// TwinCAT 3 PLC project MONETRoof
// Title: MONET Roof
// Company: Georg-August-Universitaet Goettingen
// ProjectVersion: 1.1.5
// ProgramVersion: 3.1.4026.11
// libraries:
//   Tc2_Standard, * (Beckhoff Automation GmbH)
//   Tc2_System, * (Beckhoff Automation GmbH)
//   Tc3_Module, * (Beckhoff Automation GmbH)
//   BROTLib,newest,BROT
//   VisuSymbols,3.5.10.0,System
// project tree:
//   / GlobalTextList.TcGTLO, VisualizationManager.TcVMO (not stored)
//   POUs/ FB_Roof.TcPOU, FB_RoofControl.TcPOU, FB_RoofMotor.TcPOU, FB_Ramp.TcPOU
//   VISUs/ Roof.TcVIS
//   GVLs/ Global_Version.TcGVL

// ---- GVLs/Global_Version.TcGVL
{attribute 'qualified_only'}
VAR_GLOBAL CONSTANT
	// Mirrors Beckhoff's own Global_Version.stLibVersion_* pattern (see ST_LibVersion),
	// which only covers Tc2_*/Tc3_* library references, not custom ones -- until now: this
	// GVL uses Beckhoff's own naming exactly, so it merges into a consumer's Global_Version.
	// Kept in sync with <ProjectVersion> in MonetRoof.plcproj at release time.
	stLibVersion_MONETRoof : ST_LibVersion := (
		iMajor := 1,
		iMinor := 1,
		iBuild := 5,
		iRevision := 0,
		nFlags := 1,
		sVersion := '1.1.5'
	);
END_VAR

// ---- POUs/FB_Roof.TcPOU
FUNCTION_BLOCK FB_Roof
VAR_INPUT
	roof_number				: UINT;		// number of roof
	min_speed				: UINT;		// minimum speed to drive
	max_speed				: UINT;		// maximum speed to drive
	acceleration			: UINT;		// acceleration [speed/call]: the ramp time depends on the task cycle time (10 ms in all projects)
	min_position			: INT;		// minimum position of roof
	max_position			: INT;		// maximum position of roof
	max_position_diff		: INT;		// position difference between the two drives of the roof at which sync_error / limit_error trigger (smaller is tolerated)
	overtravel_margin		: INT := 10;	// stop if a drive counts more than this beyond min/max_position, e.g. with failed limit switches
	stall_timeout			: TIME := T#10S;	// stop if a drive is driven this long without a counter edge (see FB_RoofMotor)
	limit_slowdown			: REAL := 5;	// linear slowdown when moving towards limits starting at <x% and >(100-x)%
	comm					: I_Comm;
	reset_roof				: BOOL;

	slow_open				: BOOL := FALSE;	// open at min_speed, ignoring all errors and other commands
	slow_close				: BOOL := FALSE;	// close at min_speed, ignoring all errors and other commands
	
	zero_counter			: BOOL := FALSE;	// reset position counter of both motors to zero
END_VAR
VAR_OUTPUT
	sync_error				: BOOL;
	limit_error				: BOOL;
	overtravel_error		: BOOL;
	stall_error				: BOOL;
	drive_error				: BOOL;
	config_error			: BOOL;		// invalid parameters (speed / position range, max_position_diff, acceleration): the roof is held at 0
	state					: E_RoofState := E_RoofState.unknown;
	percent_open			: REAL;
	is_open					: BOOL;		// fully open (both open limit switches)
	is_closed				: BOOL;		// fully closed (both closed limit switches)
END_VAR
VAR_OUTPUT PERSISTENT
	position_valid			: BOOL;		// position counters are trustworthy: set by a limit snap, cleared by zero_counter and whenever the counters are lost
END_VAR
VAR
	// commands for roofs
	open_roof		AT%I*	: BOOL;
	close_roof		AT%I*	: BOOL;

	motors			: ARRAY[1..2] OF FB_RoofMotor;
	i				: UINT;
	
	roof_limit_open			: BOOL;		// whether any open limit switch for this roof is triggered
	roof_limit_closed		: BOOL;		// whether any close limit switch for this roof is triggered
	
	opened_event			: FB_EventLog;	// event for opened roof half
	closed_event			: FB_EventLog;	// event for closed roof half
	sync_error_event		: FB_EventLog;	// event for sync error
	limit_error_event		: FB_EventLog;	// event for limit error
	overtravel_error_event	: FB_EventLog;	// event for over-travel error
	stall_error_event		: FB_EventLog;	// event for stall error
	config_error_event		: FB_EventLog;	// event for configuration error
	
	// speed
	vel_ramp				: FB_Ramp;
	target_speed			: INT;	
	limit_speed				: REAL;
	speed					: INT;		// move speed
	
	// opening or closing?
	is_opening				: BOOL;		// move direction
	is_closing				: BOOL;	
	
	// boot-time snap guard
	bRoofInitialized		: BOOL;
END_VAR

// parameters that would make the speed wrap in TO_INT / UINT arithmetic, divide by zero in percent_open,
// or leave the roof with a permanent sync error or without any ramp
config_error := max_speed > 32767 OR min_speed > max_speed OR max_position <= min_position OR
				max_position_diff <= 0 OR acceleration = 0;

// limit switches for this roof?
roof_limit_open   := motors[1].opened AND motors[2].opened;
roof_limit_closed := motors[1].closed AND motors[2].closed;

// ramp for roof velocity (percent_open below is still the value from the end of the previous cycle)
IF slow_open THEN
	speed := TO_INT(min_speed); 
ELSIF slow_close THEN
	speed := -TO_INT(min_speed);
ELSE
	vel_ramp(
		start		:= speed,
		target		:= target_speed,
		accel		:= acceleration,
		value		=> speed);
END_IF

// get direction
is_opening := speed > 0;
is_closing := speed < 0;

// slowdown near limits
IF is_closing AND percent_open < limit_slowdown THEN
	// closing near limit
	IF percent_open <= 0 THEN
		limit_speed := -TO_INT(min_speed);
	ELSE
		limit_speed := -((percent_open / limit_slowdown) * (max_speed - min_speed) + min_speed);
	END_IF
	IF limit_speed > speed THEN
		speed :=  REAL_TO_INT(MAX(limit_speed, -TO_INT(max_speed)));
	END_IF	
END_IF
IF is_opening AND 100.0 - percent_open < limit_slowdown THEN
	// opening near limit
	IF percent_open >= 100 THEN
		limit_speed := min_speed;
	ELSE
		limit_speed := ((100.0 - percent_open) / limit_slowdown) * (max_speed - min_speed) + min_speed;
	END_IF
	IF limit_speed < speed THEN
		speed := REAL_TO_INT(MIN(limit_speed, max_speed));
	END_IF	
END_IF

// stop on limit switches
IF (is_closing AND roof_limit_closed) OR (is_opening AND roof_limit_open) THEN
	Stop();
END_IF

// boot-time position snap: warm restart with the roof parked at a limit.
// One-shot on the first cycle, both sensors together (symmetric — no |diff|).
// Uses FB_Roof's own min_position/max_position, not motors[i].min_position/max_position: the
// latter are FB_RoofMotor's VAR_INPUTs, only assigned by the motor call further below, so on the
// very first cycle ever (before that call has run once) they are still 0.
IF NOT bRoofInitialized THEN
	bRoofInitialized := TRUE;
	// position_valid is PERSISTENT and may be stale: TwinCAT does not flush persistent data every
	// cycle, so an uncontrolled power loss mid-move can restore a value from before the roof's last
	// recorded position, with position_valid still TRUE from that earlier, once-valid state. Distrust
	// it unconditionally on every restart (clean or not, there is no way to tell them apart here) and
	// require it to be reconfirmed below, exactly like a lost/zeroed counter.
	position_valid := FALSE;
	IF roof_limit_closed THEN
		motors[1].SetPosition(min_position);
		motors[2].SetPosition(min_position);
		position_valid := TRUE;
	ELSIF roof_limit_open THEN
		motors[1].SetPosition(max_position);
		motors[2].SetPosition(max_position);
		position_valid := TRUE;
	END_IF
END_IF

// limit re-sync: snap both drives to the physical end position (both sensors
// engaged). Direction-gated: must NOT fire at the START of a move while the
// opposite limit switch is still engaged (the first counter edge can arrive
// ~0.5 s before the closed switch releases) — an ungated snap would erase
// those legitimate counts and leave the move one count short. While stalled
// against a limit the snap holds the position, so stall-jitter counts cannot
// drive it past the end position.
IF is_closing AND roof_limit_closed THEN
	motors[1].SetPosition(min_position);
	motors[2].SetPosition(min_position);
	position_valid := TRUE;
END_IF
IF is_opening AND roof_limit_open THEN
	motors[1].SetPosition(max_position);
	motors[2].SetPosition(max_position);
	position_valid := TRUE;
END_IF

// zeroing the counters says nothing about where the roof is
IF zero_counter THEN
	position_valid := FALSE;
END_IF

// latched error: hold the drive at 0 from the start of the cycle. Without this a level command
// (button held, open_roofs set) re-arms the ramp every cycle and the drive gets one ramp step
// (real_speed = acceleration) before the error stop below zeroes it again.
// Slow mode ignores errors on purpose, so it is exempted here explicitly: it must not depend
// on the motors being called before the error stop.
// A configuration error is not exempted: with invalid parameters the speed can wrap to the
// opposite direction, slow mode included.
IF config_error OR (state = E_RoofState.error AND NOT slow_open AND NOT slow_close) THEN
	Stop();
END_IF

// call motors
drive_error := FALSE;
FOR i := 1 TO 2 DO
	// call individual motors
	motors[i](
		roof_number 		:= roof_number,
		drive_number 		:= i,
		min_position 		:= min_position, 
		max_position 		:= max_position,
		real_speed			:= speed,
		zero_counter		:= zero_counter,
		stall_timeout		:= stall_timeout,
		comm 				:= comm);
		
	// check errors
	IF motors[i].error THEN
		drive_error := TRUE;
	END_IF
END_FOR
percent_open := (motors[1].percent_open + motors[2].percent_open) / 2.0;

// fully open/closed
is_open := roof_limit_open;
is_closed := roof_limit_closed;

// consistency check: no direction_error any more (removed) — the two motors of a roof half are
// always called with the same speed and are mechanically coupled by a shaft, so they can never
// disagree on direction; a mismatch between them can only ever show up as sync_error.
sync_error := ABS(motors[1].position - motors[2].position) >= max_position_diff;
limit_error := (is_opening AND motors[1].MovedSinceOpen >= max_position_diff) OR 
			   (is_closing AND motors[1].MovedSinceClosed >= max_position_diff) OR
			   (is_opening AND motors[2].MovedSinceOpen >= max_position_diff) OR 
			   (is_closing AND motors[2].MovedSinceClosed >= max_position_diff);

// no software end stop otherwise: with failed limit switches nothing bounds the travel.
// Only while the position is known: after lost/zeroed counters (e.g. a reset with the roof
// halfway open) it would block moving towards the end the counters wrongly claim to be at.
overtravel_error := position_valid AND
					((is_opening AND (motors[1].position > max_position + overtravel_margin OR 
									  motors[2].position > max_position + overtravel_margin)) OR
					 (is_closing AND (motors[1].position < min_position - overtravel_margin OR 
									  motors[2].position < min_position - overtravel_margin)));

// a drive that is driven but does not count (jam, ice, dead sensor)
stall_error := motors[1].stall_error OR motors[2].stall_error;

// stop on error
IF sync_error OR drive_error OR limit_error OR overtravel_error OR stall_error OR config_error OR state = E_RoofState.error THEN
	Stop();
END_IF

// set state
IF sync_error OR drive_error OR limit_error OR overtravel_error OR stall_error OR config_error THEN
	state := E_RoofState.error;
ELSE
	// no current error, but if we're still in error state, only proceed, if reset_roof is set
	IF state <> E_RoofState.error OR reset_roof THEN
		reset_roof := FALSE; 	

		// check other states
		// both motors get the same speed, so a moving roof has exactly one direction
		IF motors[1].moving OR motors[2].moving THEN
			IF motors[1].direction_open OR motors[2].direction_open THEN
				state := E_RoofState.opening;
			ELSE
				state := E_RoofState.closing;
			END_IF
		ELSIF roof_limit_open THEN
			// fully open needs both switches, like is_open; one switch alone is only 'stopped'
			state := E_RoofState.opened;
		ELSIF roof_limit_closed THEN
			state := E_RoofState.closed;
		ELSE
			state := E_RoofState.stopped;
		END_IF
	END_IF
END_IF

// events
opened_event(
	Trigger := is_open, 
	Level := ADSLOG_MSGTYPE_HINT, 
	FormatString := 'Roof #%s is fully open.', 
	OnMessage := UINT_TO_STRING(roof_number),
	Comm := comm);
closed_event(
	Trigger := is_closed, 
	Level := ADSLOG_MSGTYPE_HINT, 
	FormatString := 'Roof #%s is fully closed.', 
	OnMessage := UINT_TO_STRING(roof_number),
	Comm := comm); 

// errors
sync_error_event(
	Trigger := sync_error, 
	Level := ADSLOG_MSGTYPE_ERROR, 
	FormatString := 'Drives for roof #%s out of sync.', 
	OnMessage := UINT_TO_STRING(roof_number),
	Comm := comm); 
limit_error_event(
	Trigger := limit_error, 
	Level := ADSLOG_MSGTYPE_ERROR, 
	FormatString := 'Could not find 2nd limit switch for roof #%s.', 
	OnMessage := UINT_TO_STRING(roof_number),
	Comm := comm); 
overtravel_error_event(
	Trigger := overtravel_error, 
	Level := ADSLOG_MSGTYPE_ERROR, 
	FormatString := 'Roof #%s moved beyond its end position.', 
	OnMessage := UINT_TO_STRING(roof_number),
	Comm := comm); 
stall_error_event(
	Trigger := stall_error, 
	Level := ADSLOG_MSGTYPE_ERROR, 
	FormatString := 'Drive of roof #%s does not move (no counts).',
	OnMessage := UINT_TO_STRING(roof_number),
	Comm := comm);
config_error_event(
	Trigger := config_error,
	Level := ADSLOG_MSGTYPE_ERROR,
	FormatString := 'Roof #%s has invalid parameters.',
	OnMessage := UINT_TO_STRING(roof_number),
	Comm := comm);

METHOD Automatic : BOOL
VAR_INPUT
	open_roof	: BOOL;
	close_roof	: BOOL;
	stop_roof	: BOOL;
END_VAR
// automatic commands 
IF open_roof THEN
	Open();
ELSIF close_roof THEN
	Close();
ELSIF stop_roof THEN
	SoftStop();
END_IF
END_METHOD

METHOD Close : BOOL
VAR_INPUT
END_VAR
IF NOT slow_open AND NOT slow_close THEN
	IF NOT is_closed THEN
		target_speed := -TO_INT(max_speed);
	END_IF
END_IF
END_METHOD

PROPERTY Error : STRING
GET
// invalid parameters come first, the other checks are meaningless with them;
// then a drive fault: it is usually the root cause of the stall or sync error that follows
IF config_error THEN
	Error := 'Configuration error';
ELSIF drive_error THEN
	Error := 'Drive error';
ELSIF sync_error THEN
	Error := 'Sync error';
ELSIF limit_error THEN
	Error := 'Limit error';
ELSIF overtravel_error THEN
	Error := 'Over-travel error';
ELSIF stall_error THEN
	Error := 'Stall error';
ELSE
	Error := '';
END_IF
END_GET
END_PROPERTY

METHOD Manual : BOOL
VAR_INPUT
END_VAR
// manual commands commands
IF open_roof THEN
	Open();
ELSIF close_roof THEN
	Close();
ELSE
	SoftStop();
END_IF
END_METHOD

METHOD Open : BOOL
VAR_INPUT
END_VAR
VAR
END_VAR
IF NOT slow_open AND NOT slow_close THEN
	IF NOT is_open THEN
		target_speed := TO_INT(max_speed);
	END_IF
END_IF
END_METHOD

METHOD Reset : BOOL
VAR_INPUT
END_VAR
reset_roof := TRUE;
FOR i := 1 TO 2 DO
	motors[i].Reset();
END_FOR;
END_METHOD

METHOD SoftStop : BOOL
VAR_INPUT
END_VAR
target_speed := 0;
END_METHOD

PROPERTY Status : STRING
GET
IF state = E_RoofState.closed THEN
	Status := 'CLOSED';
ELSIF state = E_RoofState.opened THEN
	Status := 'OPENED';
ELSIF state = E_RoofState.opening THEN
	Status := 'OPENING';
ELSIF state = E_RoofState.closing THEN
	Status := 'CLOSING';
ELSIF state = E_RoofState.stopped THEN
	Status := 'STOPPED';
ELSIF state = E_RoofState.error THEN
	Status := 'ERROR';
ELSIF state = E_RoofState.unknown THEN
	Status := 'UNKNOWN';	
END_IF
END_GET
END_PROPERTY

METHOD Stop : BOOL
VAR_INPUT
END_VAR
speed := 0;
target_speed := 0;
END_METHOD

END_FUNCTION_BLOCK

// ---- POUs/FB_RoofMotor.TcPOU
FUNCTION_BLOCK FB_RoofMotor
VAR_INPUT
	roof_number				: UINT;		// number of roof
	drive_number			: UINT;		// number of drive
	min_position			: INT;		// minimum position of roof
	max_position			: INT;		// maximum position of roof
	real_speed				: INT;		// signed speed
	zero_counter			: BOOL := FALSE;	// reset position counter to zero
	comm					: I_Comm;
	
	// counting filters (insurance; defaults sized from the recordings — plan 2026-08-20)
	counter_debounce		: TIME := T#5MS;	// min. on-time of a sensor pulse. Keep clear of the 10 ms task cycle: at
										// PT = cycle time, ordinary cycle jitter can push the elapsed time on the
										// deciding scan just under PT and drop an otherwise-valid pulse entirely
										// (modelled in testing/check_debounce_aliasing.py). 5 ms sits above the
										// EL1008's ~3 ms input filter and comfortably below one cycle.
	counter_min_spacing		: TIME := T#50MS;	// min. time between accepted counts — keep < rotation period (600 ms)
	
	// stall watchdog
	stall_timeout			: TIME := T#10S;	// max. time moving without an accepted count — keep well above the rotation period (0.6 s at max_speed, slower at min_speed) and the ~3 s until the first count after a start
END_VAR
VAR_OUTPUT PERSISTENT
	position				: INT;	// position
END_VAR
VAR_OUTPUT
	percent_open			: REAL;	// percentage open
	
	// moving
	moving					: BOOL;
	
	// debug: raw (unfiltered, ungated) edge count for validation
	raw_counts				: DINT;
	
	// error 
	motor_error		AT%I*	: BOOL;
	error					: BOOL;
	stall_error				: BOOL;	// moving, but no counter edge for stall_timeout (jammed drive, dead sensor)
	
	// signals from limit switches
	opened			AT%I*	: BOOL;
	closed			AT%I*	: BOOL;
	
	// position on limit switch
	position_open			: INT := -1000;
	position_close			: INT := -1000;
END_VAR
VAR
	// error
	drive_error_event		: FB_EventLog;

	// inductive sensor for counting rotation
	counter			AT%I*	: BOOL;
	counter_trig			: R_TRIG;
	counter_raw_trig		: R_TRIG;	// raw (unfiltered) edge trigger — for validation only
	tonDebounce				: TON;		// level debounce for the sensor pulse
	tonSpacing				: TON;		// rate limit: min. spacing between accepted counts
	tonStall				: TON;		// time since the last accepted count while moving
	bCountAccepted			: BOOL;		// a count was accepted in this cycle
	
	// reset command to drive
	reset_command			: BOOL;
	reset_timer				: TON;
	reset_drive		AT%Q*	: BOOL;
	
	// speed
	speed			AT%Q*	: INT;		// move speed
	direction_open	AT%Q*	: BOOL;		// move direction
	direction_close	AT%Q*	: BOOL;
	
	// position on limit switch
	position_open_on_trig	: R_TRIG;
	position_open_off_trig	: F_TRIG;
	position_close_on_trig	: R_TRIG;
	position_close_off_trig	: F_TRIG;
END_VAR

// signals
error := NOT motor_error;

// reset?
//reset_timer();
IF reset_command THEN
	// set signal and start timer
	reset_drive := TRUE;
	reset_timer(IN := TRUE, PT := T#200MS);
END_IF
IF reset_timer.Q THEN
	// reset everything
	reset_drive := FALSE;
	reset_command := FALSE;
	reset_timer(IN := FALSE);
END_IF

// relative position; FB_Roof still calls the motors with max_position <= min_position when config_error is set,
// and a division by zero stops the user-mode runtime (STATUS_FLOAT_DIVIDE_BY_ZERO)
IF max_position > min_position THEN
	percent_open := 1.0 * (position - min_position) / (max_position - min_position) * 100.0;
ELSE
	percent_open := 0.0;
END_IF

// get direction
direction_open := real_speed > 0;
direction_close := real_speed < 0;

// set moving before the counter gate (motion gate: no counting while idle)
moving := real_speed <> 0;

// counter for position — filtered and gated.
// The limit re-sync in FB_Roof is the primary protection; these layers are
// insurance only. Deliberately NOT gated on the limit switches: that would
// blind the sync check to a broken connection or a stalled drive.
tonDebounce(IN := counter, PT := counter_debounce);	// stable-high filter (kills short glitches)
counter_trig(CLK := tonDebounce.Q);					// edge of the filtered signal

// raw edge count (unfiltered, ungated) — for validation/comparison
counter_raw_trig(CLK := counter);
IF counter_raw_trig.Q THEN
	raw_counts := raw_counts + 1;
END_IF

bCountAccepted := FALSE;
IF counter_trig.Q AND moving THEN					// motion gate
	IF tonSpacing.Q THEN							// spacing window since last accepted count elapsed -> accept
		tonSpacing(IN := FALSE);					// restart the spacing window
		bCountAccepted := TRUE;
		IF direction_open THEN
			position := position + 1;
		ELSIF direction_close THEN
			position := position - 1;
		END_IF
	END_IF
END_IF
tonSpacing(IN := TRUE, PT := counter_min_spacing);	// rate limit timer (runs continuously)

// stall watchdog: driven, but the position counter does not advance (both drives jammed
// gives no position difference, so sync_error cannot see it)
tonStall(IN := moving AND NOT bCountAccepted, PT := stall_timeout);
stall_error := tonStall.Q;

// zero?
IF zero_counter THEN
	position := 0;
	raw_counts := 0;
END_IF

// remember position when entering/leaving limit switches
position_open_on_trig(CLK := opened);
IF position_open_on_trig.Q THEN
	position_open := position;
END_IF
position_open_off_trig(CLK := opened);
IF position_open_off_trig.Q THEN
	position_open := -1000;
END_IF
position_close_on_trig(CLK := closed);
IF position_close_on_trig.Q THEN
	position_close := position;
END_IF
position_close_off_trig(CLK := closed);
IF position_close_off_trig.Q THEN
	position_close := -1000;
END_IF

// absolute speed
speed := ABS(real_speed);

// error
drive_error_event(	
	Trigger 		:= error, 
	Level 			:= ADSLOG_MSGTYPE_ERROR,
	FormatString 	:= 'Drive %s in error state.', 
	OnMessage 		:= CONCAT(CONCAT(CONCAT('#', UINT_TO_STRING(drive_number)), ' of roof #'), UINT_TO_STRING(roof_number)),
	Comm			:= comm);

PROPERTY MovedSinceClosed : INT
GET
IF position_close = -1000 THEN
	MovedSinceClosed := 0;
ELSE
	MovedSinceClosed := ABS(position - position_close);
END_IF
END_GET
END_PROPERTY

PROPERTY MovedSinceOpen : INT
GET
IF position_open = -1000 THEN
	MovedSinceOpen := 0;
ELSE
	MovedSinceOpen := ABS(position - position_open);
END_IF
END_GET
END_PROPERTY

METHOD Reset : BOOL
VAR_INPUT
END_VAR
reset_command := TRUE;
END_METHOD

METHOD SetPosition : BOOL
VAR_INPUT
	position_value		: INT;		// new position value (e.g. min/max_position on limit re-sync)
END_VAR
// 'position' is a VAR_OUTPUT — read-only from outside the FB, so the
// FB_Roof-level limit re-sync sets it through this method.
position := position_value;

// Re-anchor the limit-switch records of a switch that is engaged right now. They hold the counter
// reading at engagement, which is meaningless after the snap (e.g. a restart with the roof half
// open: the switch engages at a wrong reading, the snap then corrects the counter). Left alone,
// MovedSince* would report the correction as travel and raise a false limit_error.
// A drive that really overruns its switch still trips limit_error: that check runs every cycle
// before a snap can happen, and a snap needs both switches engaged.
IF opened THEN
	position_open := position_value;
END_IF
IF closed THEN
	position_close := position_value;
END_IF
END_METHOD

END_FUNCTION_BLOCK

// ---- POUs/FB_Ramp.TcPOU
FUNCTION_BLOCK FB_Ramp
VAR_INPUT
	start	: INT;
	target	: INT;
	accel	: UINT;
END_VAR
VAR_OUTPUT
	value	: INT;
END_VAR
VAR
END_VAR

value := start;

// step
// compare in DINT: a reversal (e.g. -30000 -> +30000) does not fit in 16 bit
IF TO_DINT(target) - TO_DINT(value) > 0 THEN	
	value := value + TO_INT(accel);
	IF value >= target THEN
		value := target;
	END_IF
ELSE
	value := value - TO_INT(accel);
	IF value <= target THEN
		value := target;
	END_IF
END_IF

END_FUNCTION_BLOCK

// ---- POUs/FB_RoofControl.TcPOU
FUNCTION_BLOCK FB_RoofControl IMPLEMENTS I_Roof
VAR_INPUT
	min_speed				: UINT;			// minimum speed to drive
	max_speed				: UINT;			// maximum speed to drive
	acceleration			: UINT;			// acceleration [speed/call]
	max_position_diff		: INT;			// position difference between the two drives of a roof at which sync_error / limit_error trigger (smaller is tolerated)
	limit_slowdown			: REAL := 5;	// linear slowdown when moving towards limits starting at <x% and >(100-x)%
	min_position_1			: INT := 0;		// minimum position of roof
	max_position_1			: INT := 200;		// maximum position of roof
	min_position_2			: INT := 0;		// minimum position of roof
	max_position_2			: INT := 200;		// maximum position of roof

	// commands for automatic roof controls
	open_roofs				: BOOL;
	close_roofs				: BOOL;
	stop_roofs				: BOOL;
	reset_roofs				: BOOL;	
	open_roof				: ARRAY[1..2] OF BOOL;
	close_roof				: ARRAY[1..2] OF BOOL;
	stop_roof				: ARRAY[1..2] OF BOOL;
	reset_roof				: ARRAY[1..2] OF BOOL;
	
	// automatic mode
	automatic		AT%I*	: BOOL;
	
	// UPS failure: linked to the UPS input in the consumer projects (tsproj), not evaluated yet
	ups_fail		AT%I*	: BOOL;
	
	// telemetry interval
	fTelemetryInterval		: TIME := T#5S;
END_VAR
VAR_OUTPUT
	// state
	roof_state				: E_RoofState;
	percent_open			: REAL;	
END_VAR
VAR
	// roofs
	roofs					: ARRAY[1..2] OF FB_Roof;
	
	// loop variable	
	i						: UINT;
	
	// open and close delays
	tonOpen2Delay			: TON;
	tonClose1Delay			: TON;
	
	// Comm
	fbComm					: I_Comm;	
	tonComm 				: TON;
	
	min_positions			: ARRAY[1..2] OF INT;		// minimum position of roof
	max_positions			: ARRAY[1..2] OF INT;		// maximum position of roof
END_VAR

// min_max
min_positions[1] := min_position_1;
max_positions[1] := max_position_1;
min_positions[2] := min_position_2;
max_positions[2] := max_position_2;

// call roofs
FOR i := 1 TO 2 DO
	// reset
	IF reset_roofs OR reset_roof[i] THEN
		roofs[i].Reset();
	END_IF	

	// automatic or manual mode
	IF automatic THEN
		roofs[i].Automatic(open_roof := open_roofs OR open_roof[i], close_roof := close_roofs OR close_roof[i], stop_roof := stop_roofs OR stop_roof[i]);
	ELSE
		roofs[i].Manual();
	END_IF

	// run 
	roofs[i](		
		roof_number			:= i,
		min_speed			:= min_speed,
		max_speed 			:= max_speed, 
		acceleration 		:= acceleration, 
		min_position 		:= min_positions[i], 
		max_position 		:= max_positions[i],
		max_position_diff 	:= max_position_diff,
		limit_slowdown		:= limit_slowdown,
		comm 				:= fbComm
	);
END_FOR

// set state
IF roofs[1].state = E_RoofState.error OR roofs[2].state = E_RoofState.error THEN
	roof_state := E_RoofState.error;
ELSIF roofs[1].state = E_RoofState.opened AND roofs[2].state = E_RoofState.opened THEN
	roof_state := E_RoofState.opened;
ELSIF roofs[1].state = E_RoofState.closed AND roofs[2].state = E_RoofState.closed THEN
	roof_state := E_RoofState.closed;
ELSIF roofs[1].state = E_RoofState.opening OR roofs[2].state = E_RoofState.opening THEN
	roof_state := E_RoofState.opening;	
ELSIF roofs[1].state = E_RoofState.closing OR roofs[2].state = E_RoofState.closing THEN
	roof_state := E_RoofState.closing;
ELSIF (roofs[1].state = E_RoofState.stopped OR roofs[1].state = E_RoofState.opened OR roofs[1].state = E_RoofState.closed) AND 
      (roofs[2].state = E_RoofState.stopped OR roofs[2].state = E_RoofState.opened OR roofs[2].state = E_RoofState.closed) THEN
	roof_state := E_RoofState.stopped;
ELSE
	roof_state := E_RoofState.error;	
END_IF

// percent open, clamped to 0..100: the over-travel margin and unsynced counters (after a restart with
// the roof halfway open) let the raw value leave that range, and telemetry uses -1.0 as the error marker.
// The per-roof values stay raw as a diagnostic of the counters.
percent_open := MAX(0.0, MIN(100.0, (roofs[1].percent_open + roofs[2].percent_open) / 2.0));

// send telemetry
tonComm(IN:=TRUE, PT:=fTelemetryInterval);
IF tonComm.Q THEN // publish new payload every fTelemetryInterval (default 5 seconds)
	tonComm(IN:=FALSE);
	THIS^._SendTelemetry();	
END_IF

METHOD _SendTelemetry : BOOL
VAR_INPUT
END_VAR
IF roof_state = E_RoofState.opened THEN
	fbComm.Publish('telescope', 'dome', 'AUXILIARY.DOME.REALPOS', '1.0');
ELSIF roof_state = E_RoofState.closed THEN
	fbComm.Publish('telescope', 'dome', 'AUXILIARY.DOME.REALPOS', '0.0');
ELSIF roof_state = E_RoofState.error THEN
	fbComm.Publish('telescope', 'dome', 'AUXILIARY.DOME.REALPOS', '-1.0');
ELSE
	fbComm.Publish('telescope', 'dome', 'AUXILIARY.DOME.REALPOS', LREAL_TO_STRING(percent_open / 100.0));
END_IF

IF roof_state = E_RoofState.opened OR roof_state = E_RoofState.opening THEN
	fbComm.Publish('telescope', 'dome', 'AUXILIARY.DOME.TARGETPOS', '1.0');
ELSIF roof_state = E_RoofState.closed OR roof_state = E_RoofState.closing THEN
	fbComm.Publish('telescope', 'dome', 'AUXILIARY.DOME.TARGETPOS', '0.0');
ELSIF roof_state = E_RoofState.stopped THEN
	fbComm.Publish('telescope', 'dome', 'AUXILIARY.DOME.TARGETPOS', LREAL_TO_STRING(percent_open / 100.0));
ELSE
	fbComm.Publish('telescope', 'dome', 'AUXILIARY.DOME.TARGETPOS', '-1.0');
END_IF

IF roof_state = E_RoofState.error THEN
	fbComm.Publish('telescope', 'dome', 'AUXILIARY.DOME.ERROR_STATE', '1');
	fbComm.Publish('telescope', 'dome', 'AUXILIARY.DOME.READY_STATE', '-1.0');
ELSE
	fbComm.Publish('telescope', 'dome', 'AUXILIARY.DOME.ERROR_STATE', '0');
	IF roof_state = E_RoofState.closed THEN
		fbComm.Publish('telescope', 'dome', 'AUXILIARY.DOME.READY_STATE', '0.0');
	ELSE
		fbComm.Publish('telescope', 'dome', 'AUXILIARY.DOME.READY_STATE', '1.0');
	END_IF
END_IF

IF state = E_RoofState.opening OR state = E_RoofState.closing THEN
	fbComm.Publish('telescope', 'dome', 'AUXILIARY.DOME.MOTION_STATE', '1.0');
ELSE
	fbComm.Publish('telescope', 'dome', 'AUXILIARY.DOME.MOTION_STATE', '0.0');
END_IF

// MONET specific
fbComm.Publish('telescope', 'dome', 'MONET.ROOF.STATE', Status);
fbComm.Publish('telescope', 'dome', 'MONET.ROOF.POS1', LREAL_TO_STRING(roofs[1].percent_open));
fbComm.Publish('telescope', 'dome', 'MONET.ROOF.STATE1', roofs[1].Status);
fbComm.Publish('telescope', 'dome', 'MONET.ROOF.ERROR1', roofs[1].Error);
fbComm.Publish('telescope', 'dome', 'MONET.ROOF.POS2', LREAL_TO_STRING(roofs[2].percent_open));
fbComm.Publish('telescope', 'dome', 'MONET.ROOF.STATE2', roofs[2].Status);
fbComm.Publish('telescope', 'dome', 'MONET.ROOF.ERROR2', roofs[2].Error);
END_METHOD

METHOD Close : BOOL
VAR_INPUT
END_VAR
FOR i := 1 TO 2 DO
	roofs[i].Close();
END_FOR;
END_METHOD

//FB_Init is always available implicitly and it is used primarily for initialization.
//The return value is not evaluated. For a specific influence, you can also declare the
//methods explicitly and provide additional code there with the standard initialization
//code. You can evaluate the return value.
METHOD FB_Init: BOOL
VAR_INPUT
    bInitRetains	: BOOL; // TRUE: the retain variables are initialized (reset warm / reset cold)
    bInCopyCode		: BOOL;  // TRUE: the instance will be copied to the copy code afterward (online change)
	comm			: I_Comm;   
END_VAR
THIS^.fbComm := comm;
END_METHOD

METHOD Open : BOOL
VAR_INPUT
END_VAR
FOR i := 1 TO 2 DO
	roofs[i].Open();
END_FOR;
END_METHOD

METHOD Reset : BOOL
VAR_INPUT
END_VAR
FOR i := 1 TO 2 DO
	roofs[i].Reset();
END_FOR;
END_METHOD

PROPERTY State : E_RoofState
GET
State := roof_state;
END_GET
END_PROPERTY

PROPERTY Status : STRING
GET
IF state = E_RoofState.closed THEN
	Status := 'CLOSED';
ELSIF state = E_RoofState.opened THEN
	Status := 'OPENED';
ELSIF state = E_RoofState.opening THEN
	Status := 'OPENING';
ELSIF state = E_RoofState.closing THEN
	Status := 'CLOSING';
ELSIF state = E_RoofState.stopped THEN
	Status := 'STOPPED';
ELSIF state = E_RoofState.error THEN
	Status := 'ERROR';
ELSIF state = E_RoofState.unknown THEN
	Status := 'UNKNOWN';	
END_IF
END_GET
END_PROPERTY

METHOD Stop : BOOL
VAR_INPUT
END_VAR
FOR i := 1 TO 2 DO
	roofs[i].Stop();
END_FOR;
END_METHOD

END_FUNCTION_BLOCK

// ---- GlobalTextList.TcGTLO
TEXTLIST GlobalTextList
  265 = '%.0f %'
  194 = '%.2f'
  616 = '%d'
  606 = '%d %'
  759 = '%d %%'
  792 = '%s'
  148 = 'Automatic'
  337 = 'Close'
  507 = 'Closed'
  272 = 'Closing'
  937 = 'Dir Error'
  59 = 'Directio n Error'
  475 = 'Direction Error'
  957 = 'Direction error'
  511 = 'Drive   Error'
  264 = 'DriveError'
  298 = 'Error'
  389 = 'Motor #1'
  611 = 'Motor #2'
  765 = 'Moving'
  576 = 'None'
  366 = 'Open'
  186 = 'Opening'
  523 = 'Position'
  375 = 'Reset'
  798 = 'Roof'
  456 = 'Roof #1'
  944 = 'Roof #2'
  138 = 'Slow close'
  996 = 'Slow open'
  49 = 'Speed'
  520 = 'State'
  838 = 'Stop'
  790 = 'Stopped'
  619 = 'Sync Error'
  385 = 'Sync error'
  609 = 'Zero counter'
END_TEXTLIST

// ---- VISUs/Roof.TcVIS
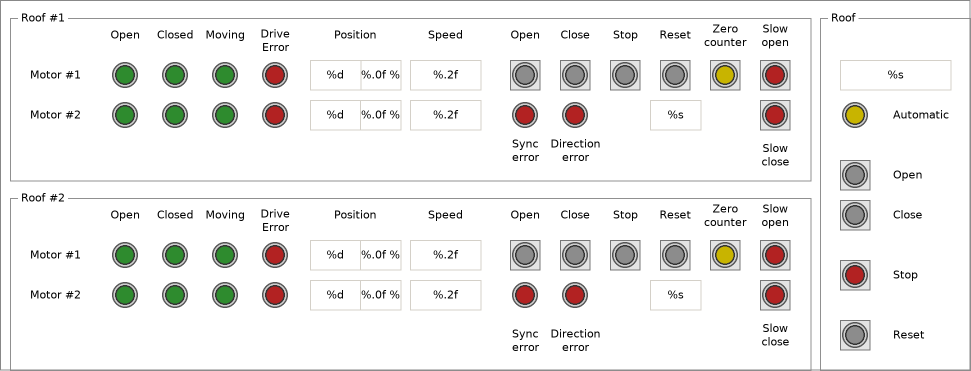
VISUALIZATION Roof  // 971x371
    GroupBox (10,10 801x171), "Roof #1"
        Label (10,50 71x30), "Motor #1"
        Label (10,90 71x30), "Motor #2"
        Label (80,10 71x30), "Open"
        Label (130,10 71x30), "Closed"
        Lamp1 (100,50 30x30), variable: MAIN.RoofControl.roofs[1].motors[1].opened, style: Lamp-Lamp1-Green
        Lamp1 (150,50 30x30), variable: MAIN.RoofControl.roofs[1].motors[1].closed, style: Lamp-Lamp1-Green
        Lamp1 (100,90 30x30), variable: MAIN.RoofControl.roofs[1].motors[2].opened, style: Lamp-Lamp1-Green
        Lamp1 (150,90 30x30), variable: MAIN.RoofControl.roofs[1].motors[2].closed, style: Lamp-Lamp1-Green
        Label (180,10 71x30), "Moving"
        Lamp1 (200,50 30x30), variable: MAIN.RoofControl.roofs[1].motors[1].moving, style: Lamp-Lamp1-Green
        Lamp1 (200,90 30x30), variable: MAIN.RoofControl.roofs[1].motors[2].moving, style: Lamp-Lamp1-Green
        Label (310,10 71x30), "Position"
        Textfield (350,50 41x30), "%.0f %", text variable: MAIN.RoofControl.roofs[1].motors[1].percent_open, input disabled if: TRUE
        Textfield (300,90 51x30), "%d", text variable: MAIN.RoofControl.roofs[1].motors[2].position, input disabled if: TRUE
        Label (400,10 71x30), "Speed"
        Textfield (400,50 71x30), "%.2f", text variable: MAIN.RoofControl.roofs[1].motors[1].speed, input disabled if: TRUE
        Textfield (400,90 71x30), "%.2f", text variable: MAIN.RoofControl.roofs[1].motors[2].speed, input disabled if: TRUE
        Label (480,10 71x30), "Open"
        PushSwitch (500,50 30x30), variable: MAIN.RoofControl.open_roof[1], behaviour: TAP, style: Switch-PushSwitch-Gray
        PushSwitch (550,50 30x30), variable: MAIN.RoofControl.close_roof[1], behaviour: TAP, style: Switch-PushSwitch-Gray
        Label (530,10 71x30), "Close"
        Label (590,10 51x30), "Stop"
        PushSwitch (600,50 30x30), variable: MAIN.RoofControl.stop_roof[1], behaviour: TAP, style: Switch-PushSwitch-Gray
        Lamp1 (500,90 30x30), variable: MAIN.RoofControl.roofs[1].sync_error, style: Lamp-Lamp1-Red
        Textfield (640,90 51x30), "%s", text variable: MAIN.RoofControl.roofs[1].state, input disabled if: TRUE
        Textfield (300,50 51x30), "%d", text variable: MAIN.RoofControl.roofs[1].motors[1].position, input disabled if: TRUE
        Textfield (350,90 41x30), "%.0f %", text variable: MAIN.RoofControl.roofs[1].motors[2].percent_open, input disabled if: TRUE
        Label (240,10 51x41), "Drive Error"
        Lamp1 (550,90 30x30), variable: MAIN.RoofControl.roofs[1].direction_error, style: Lamp-Lamp1-Red
        Label (490,120 51x41), "Sync error"
        Label (530,120 71x41), "Direction error"
        Label (640,10 51x30), "Reset"
        Lamp1 (250,50 30x30), variable: MAIN.RoofControl.roofs[1].motors[1].error, style: Lamp-Lamp1-Red
        Lamp1 (250,90 30x30), variable: MAIN.RoofControl.roofs[1].motors[2].error, style: Lamp-Lamp1-Red
        PushSwitch (750,50 30x30), variable: MAIN.RoofControl.roofs[1].slow_open, behaviour: TAP, style: Switch-PushSwitch-Red
        Label (740,10 51x31), "Slow open"
        Label (740,130 51x30), "Slow close"
        PushSwitch (750,230 30x30), variable: MAIN.RoofControl.stop_roof[1], behaviour: TAP, style: Switch-PushSwitch-Gray
        Label (690,10 51x31), "Zero counter"
    GroupBox (10,190 801x181), "Roof #2"
        Label (10,50 71x30), "Motor #1"
        Label (10,90 71x30), "Motor #2"
        Label (80,10 71x30), "Open"
        Label (130,10 71x30), "Closed"
        Lamp1 (100,50 30x30), variable: MAIN.RoofControl.roofs[2].motors[1].opened, style: Lamp-Lamp1-Green
        Lamp1 (150,50 30x30), variable: MAIN.RoofControl.roofs[2].motors[1].closed, style: Lamp-Lamp1-Green
        Lamp1 (100,90 30x30), variable: MAIN.RoofControl.roofs[2].motors[2].opened, style: Lamp-Lamp1-Green
        Lamp1 (150,90 30x30), variable: MAIN.RoofControl.roofs[2].motors[2].closed, style: Lamp-Lamp1-Green
        Label (180,10 71x30), "Moving"
        Lamp1 (200,50 30x30), variable: MAIN.RoofControl.roofs[2].motors[1].moving, style: Lamp-Lamp1-Green
        Lamp1 (200,90 30x30), variable: MAIN.RoofControl.roofs[2].motors[2].moving, style: Lamp-Lamp1-Green
        Label (310,10 71x30), "Position"
        Textfield (300,50 51x30), "%d", text variable: MAIN.RoofControl.roofs[2].motors[1].position, input disabled if: TRUE
        Textfield (300,90 51x30), "%d", text variable: MAIN.RoofControl.roofs[2].motors[2].position, input disabled if: TRUE
        Label (400,10 71x30), "Speed"
        Textfield (400,50 71x30), "%.2f", text variable: MAIN.RoofControl.roofs[2].motors[1].speed, input disabled if: TRUE
        Textfield (400,90 71x30), "%.2f", text variable: MAIN.RoofControl.roofs[2].motors[2].speed, input disabled if: TRUE
        Label (480,10 71x30), "Open"
        PushSwitch (500,50 30x30), variable: MAIN.RoofControl.open_roof[2], behaviour: TAP, style: Switch-PushSwitch-Gray
        PushSwitch (550,50 30x30), variable: MAIN.RoofControl.close_roof[2], behaviour: TAP, style: Switch-PushSwitch-Gray
        Label (530,10 71x30), "Close"
        Label (590,10 51x30), "Stop"
        PushSwitch (600,50 30x30), variable: MAIN.RoofControl.stop_roof[2], behaviour: TAP, style: Switch-PushSwitch-Gray
        Lamp1 (500,90 30x30), variable: MAIN.RoofControl.roofs[2].sync_error, style: Lamp-Lamp1-Red
        Textfield (640,90 51x30), "%s", text variable: MAIN.RoofControl.roofs[2].state, input disabled if: TRUE
        Textfield (350,50 41x30), "%.0f %", text variable: MAIN.RoofControl.roofs[2].motors[1].percent_open, input disabled if: TRUE
        Textfield (350,90 41x30), "%.0f %", text variable: MAIN.RoofControl.roofs[2].motors[2].percent_open, input disabled if: TRUE
        Label (240,10 51x41), "Drive Error"
        Label (490,130 51x41), "Sync error"
        Label (530,130 71x41), "Direction error"
        Lamp1 (550,90 30x30), variable: MAIN.RoofControl.roofs[2].direction_error, style: Lamp-Lamp1-Red
        Lamp1 (250,90 30x30), variable: MAIN.RoofControl.roofs[2].motors[2].error, style: Lamp-Lamp1-Red
        Lamp1 (250,50 30x30), variable: MAIN.RoofControl.roofs[2].motors[1].error, style: Lamp-Lamp1-Red
        PushSwitch (750,50 30x30), variable: MAIN.RoofControl.roofs[2].slow_open, behaviour: TAP, style: Switch-PushSwitch-Red
        PushSwitch (750,90 30x30), variable: MAIN.RoofControl.stop_roof[1], behaviour: TAP, style: Switch-PushSwitch-Gray
        PushSwitch (750,-90 30x30), variable: MAIN.RoofControl.stop_roof[1], behaviour: TAP, style: Switch-PushSwitch-Gray
        Label (740,130 51x30), "Slow close"
        Label (690,10 51x31), "Zero counter"
    GroupBox (820,10 151x361), "Roof"
        Label (70,150 71x30), "Open"
        PushSwitch (20,150 30x30), variable: MAIN.RoofControl.open_roofs, behaviour: TAP, style: Switch-PushSwitch-Gray
        PushSwitch (20,190 30x30), variable: MAIN.RoofControl.close_roofs, behaviour: TAP, style: Switch-PushSwitch-Gray
        Label (70,190 71x30), "Close"
        Label (70,250 71x30), "Stop"
        PushSwitch (20,250 30x30), variable: MAIN.RoofControl.stop_roofs, behaviour: TAP, style: Switch-PushSwitch-Red
        Label (70,90 71x30), "Automatic"
        Lamp1 (20,90 30x30), variable: MAIN.RoofControl.automatic, style: Lamp-Lamp1-Yellow
        Label (70,310 71x30), "Reset"
        PushSwitch (20,310 30x30), variable: MAIN.RoofControl.reset_roofs, behaviour: TAP, style: Switch-PushSwitch-Gray
        Textfield (20,50 111x30), "%s", text variable: MAIN.RoofControl.roofs[1].state, input disabled if: TRUE
    PushSwitch (660,60 30x30), variable: MAIN.RoofControl.reset_roof[1], behaviour: TAP, style: Switch-PushSwitch-Gray
    Label (650,200 51x30), "Reset"
    PushSwitch (660,240 30x30), variable: MAIN.RoofControl.reset_roof[2], behaviour: TAP, style: Switch-PushSwitch-Gray
    PushSwitch (710,60 30x30), variable: MAIN.RoofControl.roofs[1].zero_counter, behaviour: TAP, style: Switch-PushSwitch-Yellow
    Label (750,200 51x31), "Slow open"
    PushSwitch (710,240 30x30), variable: MAIN.RoofControl.roofs[2].zero_counter, behaviour: TAP, style: Switch-PushSwitch-Yellow
    PushSwitch (760,280 30x30), variable: MAIN.RoofControl.roofs[2].slow_close, behaviour: TAP, style: Switch-PushSwitch-Red
    PushSwitch (760,100 30x30), variable: MAIN.RoofControl.roofs[1].slow_close, behaviour: TAP, style: Switch-PushSwitch-Red
END_VISUALIZATION
